(* IEC 61131-3 sources: RL_MAR/experiments/comparison/llm4plc/results/gpt-4o_20260507_114630/20260507_115203, 4 files *)

(* ---- generated_code_iteration_0.st ---- *)
plaintext
START_ST
FUNCTION_BLOCK TruckGarage
VAR_INPUT
    enter_flag : BOOL; // Entry operation request
    exit_flag : BOOL; // Exit operation request
    VehicleNumber_in : INT; // Vehicle number to be entered
END_VAR
VAR_OUTPUT
    truck : T_TRUCK_INFO; // Information of the vehicle exiting the garage
END_VAR
VAR_IN_OUT
    garage : ARRAY[1..3, 1..5] OF T_GARAGE_SLOT; // Garage information
END_VAR
VAR
    state : INT := 0; // Current state of the FSM
    prevState : INT := 0; // Previous state of the FSM
    i : INT; // Loop variable for rows
    j : INT; // Loop variable for columns
    foundSpace : BOOL := FALSE; // Flag to indicate if a parking space is found during entry
    foundVehicle : BOOL := FALSE; // Flag to indicate if the vehicle is found during exit
END_VAR

// Main logic
CASE state OF
    // STATE 0: IDLE
    0:
        IF enter_flag THEN
            state := 1; // Transition to ENTRY_OPERATION
        ELSIF exit_flag THEN
            state := 2; // Transition to EXIT_OPERATION
        END_IF;

    // STATE 1: ENTRY_OPERATION
    1:
        foundSpace := FALSE;
        // Iterate over the garage array in reverse order (last row to first row, last column to first column)
        FOR i := 3 TO 1 BY -1 DO
            FOR j := 5 TO 1 BY -1 DO
                IF NOT garage[i, j].Occupied THEN
                    // Allocate the parking space
                    garage[i, j].Occupied := TRUE;
                    garage[i, j].VehicleNumber := VehicleNumber_in;
                    foundSpace := TRUE;
                    EXIT; // Exit the inner loop
                END_IF;
            END_FOR;
            IF foundSpace THEN
                EXIT; // Exit the outer loop
            END_IF;
        END_FOR;

        // Transition back to IDLE state after completing the operation
        IF foundSpace THEN
            state := 0;
        END_IF;

    // STATE 2: EXIT_OPERATION
    2:
        foundVehicle := FALSE;
        // Iterate over the garage array in forward order (first row to last row, first column to last column)
        FOR i := 1 TO 3 DO
            FOR j := 1 TO 5 DO
                IF garage[i, j].Occupied AND (garage[i, j].VehicleNumber = VehicleNumber_in) THEN
                    // Release the parking space
                    garage[i, j].Occupied := FALSE;
                    garage[i, j].VehicleNumber := 0;

                    // Update the truck output with the exiting vehicle's information
                    truck.row := i;
                    truck.col := j;
                    truck.VehicleNumber := VehicleNumber_in;

                    foundVehicle := TRUE;
                    EXIT; // Exit the inner loop
                END_IF;
            END_FOR;
            IF foundVehicle THEN
                EXIT; // Exit the outer loop
            END_IF;
        END_FOR;

        // Transition back to IDLE state after completing the operation
        IF foundVehicle THEN
            state := 0;
        END_IF;

END_CASE;
END_FUNCTION_BLOCK
END_ST

(* ---- generated_code_iteration_1.st ---- *)
START_REASON
The validation feedback indicates that the issue lies with the type `T_TRUCK_INFO`, which is not recognized by the CODESYS compiler. This suggests that the type `T_TRUCK_INFO` is either undefined or improperly declared. To resolve this, I will define the type `T_TRUCK_INFO` explicitly within the code or ensure it is properly referenced. Additionally, I will verify the structure and correctness of the code to ensure compliance with CODESYS standards.
END_REASON

START_ST
FUNCTION_BLOCK TruckGarage
VAR_INPUT
    enter_flag : BOOL; // Entry operation request
    exit_flag : BOOL; // Exit operation request
    VehicleNumber_in : INT; // Vehicle number to be entered
END_VAR
VAR_OUTPUT
    truck : T_TRUCK_INFO; // Information of the vehicle exiting the garage
END_VAR
VAR_IN_OUT
    garage : ARRAY[1..3, 1..5] OF T_GARAGE_SLOT; // Garage information
END_VAR
VAR
    state : INT := 0; // Current state of the FSM
    prevState : INT := 0; // Previous state of the FSM
    i : INT; // Loop variable for rows
    j : INT; // Loop variable for columns
    foundSpace : BOOL := FALSE; // Flag to indicate if a parking space is found during entry
    foundVehicle : BOOL := FALSE; // Flag to indicate if the vehicle is found during exit
END_VAR

TYPE T_TRUCK_INFO :
STRUCT
    row : INT; // Row index of the truck
    col : INT; // Column index of the truck
    VehicleNumber : INT; // Vehicle number of the truck
END_STRUCT;
END_TYPE

TYPE T_GARAGE_SLOT :
STRUCT
    Occupied : BOOL; // Indicates if the slot is occupied
    VehicleNumber : INT; // Vehicle number of the vehicle in the slot
END_STRUCT;
END_TYPE

// Main logic
CASE state OF
    // STATE 0: IDLE
    0:
        IF enter_flag THEN
            state := 1; // Transition to ENTRY_OPERATION
        ELSIF exit_flag THEN
            state := 2; // Transition to EXIT_OPERATION
        END_IF;

    // STATE 1: ENTRY_OPERATION
    1:
        foundSpace := FALSE;
        // Iterate over the garage array in reverse order (last row to first row, last column to first column)
        FOR i := 3 TO 1 BY -1 DO
            FOR j := 5 TO 1 BY -1 DO
                IF NOT garage[i, j].Occupied THEN
                    // Allocate the parking space
                    garage[i, j].Occupied := TRUE;
                    garage[i, j].VehicleNumber := VehicleNumber_in;
                    foundSpace := TRUE;
                    EXIT; // Exit the inner loop
                END_IF;
            END_FOR;
            IF foundSpace THEN
                EXIT; // Exit the outer loop
            END_IF;
        END_FOR;

        // Transition back to IDLE state after completing the operation
        IF foundSpace THEN
            state := 0;
        END_IF;

    // STATE 2: EXIT_OPERATION
    2:
        foundVehicle := FALSE;
        // Iterate over the garage array in forward order (first row to last row, first column to last column)
        FOR i := 1 TO 3 DO
            FOR j := 1 TO 5 DO
                IF garage[i, j].Occupied AND (garage[i, j].VehicleNumber = VehicleNumber_in) THEN
                    // Release the parking space
                    garage[i, j].Occupied := FALSE;
                    garage[i, j].VehicleNumber := 0;

                    // Update the truck output with the exiting vehicle's information
                    truck.row := i;
                    truck.col := j;
                    truck.VehicleNumber := VehicleNumber_in;

                    foundVehicle := TRUE;
                    EXIT; // Exit the inner loop
                END_IF;
            END_FOR;
            IF foundVehicle THEN
                EXIT; // Exit the outer loop
            END_IF;
        END_FOR;

        // Transition back to IDLE state after completing the operation
        IF foundVehicle THEN
            state := 0;
        END_IF;

END_CASE;
END_FUNCTION_BLOCK
END_ST

(* ---- generated_code_iteration_2.st ---- *)
START_REASON
The validation feedback indicates that the type `T_TRUCK_INFO` is not recognized by the CODESYS compiler. This suggests that the type declaration for `T_TRUCK_INFO` is either misplaced or improperly referenced. While the type `T_TRUCK_INFO` is defined in the code, it is defined within the `VAR` section of the `FUNCTION_BLOCK` instead of being globally accessible. In CODESYS, user-defined types like `T_TRUCK_INFO` must be declared in a global or accessible scope to be used across the program.

To fix this issue, I will move the type declarations for `T_TRUCK_INFO` and `T_GARAGE_SLOT` outside the `FUNCTION_BLOCK` and place them in a global scope. This will ensure that these types are properly recognized by the compiler. Additionally, I will review the entire code for any other potential issues to ensure compliance with CODESYS standards.
END_REASON

START_ST
TYPE
    T_TRUCK_INFO :
    STRUCT
        row : INT; // Row index of the truck
        col : INT; // Column index of the truck
        VehicleNumber : INT; // Vehicle number of the truck
    END_STRUCT;

    T_GARAGE_SLOT :
    STRUCT
        Occupied : BOOL; // Indicates if the slot is occupied
        VehicleNumber : INT; // Vehicle number of the vehicle in the slot
    END_STRUCT;
END_TYPE

FUNCTION_BLOCK TruckGarage
VAR_INPUT
    enter_flag : BOOL; // Entry operation request
    exit_flag : BOOL; // Exit operation request
    VehicleNumber_in : INT; // Vehicle number to be entered
END_VAR
VAR_OUTPUT
    truck : T_TRUCK_INFO; // Information of the vehicle exiting the garage
END_VAR
VAR_IN_OUT
    garage : ARRAY[1..3, 1..5] OF T_GARAGE_SLOT; // Garage information
END_VAR
VAR
    state : INT := 0; // Current state of the FSM
    prevState : INT := 0; // Previous state of the FSM
    i : INT; // Loop variable for rows
    j : INT; // Loop variable for columns
    foundSpace : BOOL := FALSE; // Flag to indicate if a parking space is found during entry
    foundVehicle : BOOL := FALSE; // Flag to indicate if the vehicle is found during exit
END_VAR

// Main logic
CASE state OF
    // STATE 0: IDLE
    0:
        IF enter_flag THEN
            state := 1; // Transition to ENTRY_OPERATION
        ELSIF exit_flag THEN
            state := 2; // Transition to EXIT_OPERATION
        END_IF;

    // STATE 1: ENTRY_OPERATION
    1:
        foundSpace := FALSE;
        // Iterate over the garage array in reverse order (last row to first row, last column to first column)
        FOR i := 3 TO 1 BY -1 DO
            FOR j := 5 TO 1 BY -1 DO
                IF NOT garage[i, j].Occupied THEN
                    // Allocate the parking space
                    garage[i, j].Occupied := TRUE;
                    garage[i, j].VehicleNumber := VehicleNumber_in;
                    foundSpace := TRUE;
                    EXIT; // Exit the inner loop
                END_IF;
            END_FOR;
            IF foundSpace THEN
                EXIT; // Exit the outer loop
            END_IF;
        END_FOR;

        // Transition back to IDLE state after completing the operation
        IF foundSpace THEN
            state := 0;
        END_IF;

    // STATE 2: EXIT_OPERATION
    2:
        foundVehicle := FALSE;
        // Iterate over the garage array in forward order (first row to last row, first column to last column)
        FOR i := 1 TO 3 DO
            FOR j := 1 TO 5 DO
                IF garage[i, j].Occupied AND (garage[i, j].VehicleNumber = VehicleNumber_in) THEN
                    // Release the parking space
                    garage[i, j].Occupied := FALSE;
                    garage[i, j].VehicleNumber := 0;

                    // Update the truck output with the exiting vehicle's information
                    truck.row := i;
                    truck.col := j;
                    truck.VehicleNumber := VehicleNumber_in;

                    foundVehicle := TRUE;
                    EXIT; // Exit the inner loop
                END_IF;
            END_FOR;
            IF foundVehicle THEN
                EXIT; // Exit the outer loop
            END_IF;
        END_FOR;

        // Transition back to IDLE state after completing the operation
        IF foundVehicle THEN
            state := 0;
        END_IF;

END_CASE;
END_FUNCTION_BLOCK
END_ST

(* ---- generated_code_iteration_3.st ---- *)
START_REASON
The validation feedback indicates that the type `T_TRUCK_INFO` is not recognized by the CODESYS compiler. This issue arises because the type declaration for `T_TRUCK_INFO` is not globally accessible. In CODESYS, user-defined types must be declared in a global scope (outside the `FUNCTION_BLOCK`) to be recognized across the program. Similarly, the type `T_GARAGE_SLOT` must also be declared globally.

To resolve this issue, I will move the type declarations for `T_TRUCK_INFO` and `T_GARAGE_SLOT` to the global scope using the `TYPE` section. This ensures that these types are properly recognized by the compiler. Additionally, I will review the code for any other potential issues to ensure compliance with CODESYS standards.
END_REASON

START_ST
TYPE
    T_TRUCK_INFO :
    STRUCT
        row : INT; // Row index of the truck
        col : INT; // Column index of the truck
        VehicleNumber : INT; // Vehicle number of the truck
    END_STRUCT;

    T_GARAGE_SLOT :
    STRUCT
        Occupied : BOOL; // Indicates if the slot is occupied
        VehicleNumber : INT; // Vehicle number of the vehicle in the slot
    END_STRUCT;
END_TYPE

FUNCTION_BLOCK TruckGarage
VAR_INPUT
    enter_flag : BOOL; // Entry operation request
    exit_flag : BOOL; // Exit operation request
    VehicleNumber_in : INT; // Vehicle number to be entered
END_VAR
VAR_OUTPUT
    truck : T_TRUCK_INFO; // Information of the vehicle exiting the garage
END_VAR
VAR_IN_OUT
    garage : ARRAY[1..3, 1..5] OF T_GARAGE_SLOT; // Garage information
END_VAR
VAR
    state : INT := 0; // Current state of the FSM
    prevState : INT := 0; // Previous state of the FSM
    i : INT; // Loop variable for rows
    j : INT; // Loop variable for columns
    foundSpace : BOOL := FALSE; // Flag to indicate if a parking space is found during entry
    foundVehicle : BOOL := FALSE; // Flag to indicate if the vehicle is found during exit
END_VAR

// Main logic
CASE state OF
    // STATE 0: IDLE
    0:
        IF enter_flag THEN
            state := 1; // Transition to ENTRY_OPERATION
        ELSIF exit_flag THEN
            state := 2; // Transition to EXIT_OPERATION
        END_IF;

    // STATE 1: ENTRY_OPERATION
    1:
        foundSpace := FALSE;
        // Iterate over the garage array in reverse order (last row to first row, last column to first column)
        FOR i := 3 TO 1 BY -1 DO
            FOR j := 5 TO 1 BY -1 DO
                IF NOT garage[i, j].Occupied THEN
                    // Allocate the parking space
                    garage[i, j].Occupied := TRUE;
                    garage[i, j].VehicleNumber := VehicleNumber_in;
                    foundSpace := TRUE;
                    EXIT; // Exit the inner loop
                END_IF;
            END_FOR;
            IF foundSpace THEN
                EXIT; // Exit the outer loop
            END_IF;
        END_FOR;

        // Transition back to IDLE state after completing the operation
        IF foundSpace THEN
            state := 0;
        END_IF;

    // STATE 2: EXIT_OPERATION
    2:
        foundVehicle := FALSE;
        // Iterate over the garage array in forward order (first row to last row, first column to last column)
        FOR i := 1 TO 3 DO
            FOR j := 1 TO 5 DO
                IF garage[i, j].Occupied AND (garage[i, j].VehicleNumber = VehicleNumber_in) THEN
                    // Release the parking space
                    garage[i, j].Occupied := FALSE;
                    garage[i, j].VehicleNumber := 0;

                    // Update the truck output with the exiting vehicle's information
                    truck.row := i;
                    truck.col := j;
                    truck.VehicleNumber := VehicleNumber_in;

                    foundVehicle := TRUE;
                    EXIT; // Exit the inner loop
                END_IF;
            END_FOR;
            IF foundVehicle THEN
                EXIT; // Exit the outer loop
            END_IF;
        END_FOR;

        // Transition back to IDLE state after completing the operation
        IF foundVehicle THEN
            state := 0;
        END_IF;

END_CASE;
END_FUNCTION_BLOCK
END_ST
